PROGRAM MAIN
VAR
END_VAR

END_PROGRAM

(* stored: Version 1.1.0.1
   POU MAIN: Id {3e4e8d08-70d8-4a56-bf44-5666e6a878fb} *)
